// TIA Portal project "GateTest" (V17)

(* hardware
DEVICE "HMI_1"  KTP400 Comfort
   slot 0: "HMI_1"  KTP400 Comfort  6AV2 124-2DC01-0AX0  17.0.0.0
   slot 1: "HMI_RT_1"  KTP400 Comfort  6AV2 124-2DC01-0AX0  17.0.0.0
   slot 5: "HMI_1.IE_CP_1"  PROFINET Interface  17.0.0.0
      slot 1: "PROFINET Interface_1"  PROFINET Interface
         slot 1: "Port_1"  Port
   slot 7: "HMI_1.MPI/DP_CP_1"  MPI/DP Interface  17.0.0.0
DEVICE "S7-1200 station_1"  S7-1200 Station
   slot 0: "Rack_0"  S7-1200 Rack  Rack  V1.0
   slot 1: "PLC_1"  CPU 1211C DC/DC/Rly  6ES7 211-1HE40-0XB0  V4.5
   slot 101: "CM 1241 (RS422/485)_1"  6ES7 241-1CH32-0XB0  V2.2
*)

// ===== PLC "PLC_1"  CPU 1211C DC/DC/Rly =====

VAR_GLOBAL   // PLC tag table "Default tag table"
   "System_Byte" AT %MB1 : Byte;
   "FirstScan" AT %M1.0 : Bool;
   "DiagStatusUpdate" AT %M1.1 : Bool;
   "AlwaysTRUE" AT %M1.2 : Bool;
   "AlwaysFALSE" AT %M1.3 : Bool;
   "Clock_Byte" AT %MB0 : Byte;
   "Clock_10Hz" AT %M0.0 : Bool;
   "Clock_5Hz" AT %M0.1 : Bool;
   "Clock_2.5Hz" AT %M0.2 : Bool;
   "Clock_2Hz" AT %M0.3 : Bool;
   "Clock_1.25Hz" AT %M0.4 : Bool;
   "Clock_1Hz" AT %M0.5 : Bool;
   "Clock_0.625Hz" AT %M0.6 : Bool;
   "Clock_0.5Hz" AT %M0.7 : Bool;
   "IHM_Sens_Droite" AT %M2.0 : Bool;
   "IHM_Sens_Gauche" AT %M2.1 : Bool;
   "SensDroite" AT %Q0.0 : Bool;
   "SensGauche" AT %Q0.1 : Bool;
   "Busy" AT %M10.0 : Bool;
   "IHM_REQ" AT %M2.2 : Bool;
   "NB_ENTREE" AT %MW30 : Int;
   "NB_SORTIE" AT %MW32 : Int;
   "NB_INTERIEUR" AT %MW34 : Int;
   "Registre" AT %MW36 : UInt;
END_VAR

DATA_BLOCK "Data_block_1"   // DB3
{ S7_Optimized_Access := 'FALSE' }
VERSION : 0.1
   VAR
      ResultREQ : Array[0..4] of UInt;
      Registre : UInt := 40001;
      Mode : Int := 0;
   END_VAR
BEGIN
END_DATA_BLOCK

FUNCTION "CommandeMoteur" : Void   // FC1, LAD
{ S7_Optimized_Access := 'TRUE' }
VERSION : 0.1
BEGIN

REGION Network 1
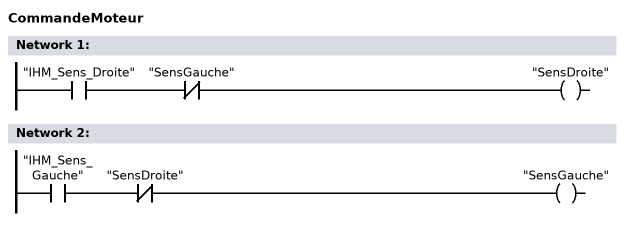
   RUNG wire#powerrail
      Contact( "IHM_Sens_Droite" )
      I_Contact( "SensGauche" )
      Coil( "SensDroite" )
   END_RUNG
   // the same network as SCL:
   "SensDroite" := "IHM_Sens_Droite" AND NOT "SensGauche";
END_REGION

REGION Network 2
   RUNG wire#powerrail
      Contact( "IHM_Sens_Gauche" )
      I_Contact( "SensDroite" )
      Coil( "SensGauche" )
   END_RUNG
   // the same network as SCL:
   "SensGauche" := "IHM_Sens_Gauche" AND NOT "SensDroite";
END_REGION
END_FUNCTION

FUNCTION "CommRS485" : Void   // FC2, LAD
{ S7_Optimized_Access := 'TRUE' }
VERSION : 0.1
BEGIN

REGION Network 1
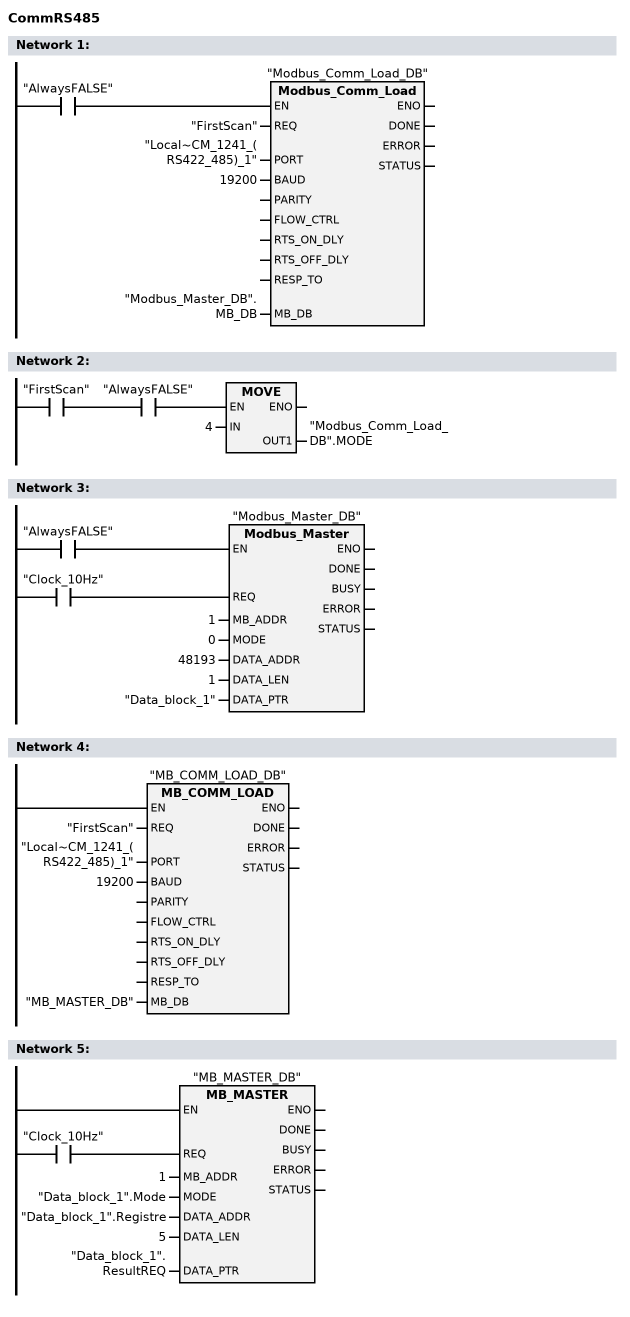
   IF "AlwaysFALSE" THEN
       "Modbus_Comm_Load_DB"(REQ := "FirstScan",   // Modbus_Comm_Load
                             PORT := "Local~CM_1241_(RS422_485)_1",
                             BAUD := 19200,
                             MB_DB := "Modbus_Master_DB".MB_DB);
   END_IF;
END_REGION

REGION Network 2
   RUNG wire#powerrail
      Contact( "FirstScan" )
      Contact( "AlwaysFALSE" )
      Move(in := 4, out1 => "Modbus_Comm_Load_DB".MODE)
   END_RUNG
   // the same network as SCL:
   IF "FirstScan" AND "AlwaysFALSE" THEN "Modbus_Comm_Load_DB".MODE := 4; END_IF;
END_REGION

REGION Network 3
   IF "AlwaysFALSE" THEN
       "Modbus_Master_DB"(REQ := "Clock_10Hz",   // Modbus_Master
                          MB_ADDR := 1,
                          MODE := 0,
                          DATA_ADDR := 48193,
                          DATA_LEN := 1,
                          DATA_PTR := "Data_block_1");
   END_IF;
END_REGION

REGION Network 4
   "MB_COMM_LOAD_DB"(REQ := "FirstScan",   // MB_COMM_LOAD
                     PORT := "Local~CM_1241_(RS422_485)_1",
                     BAUD := 19200,
                     MB_DB := "MB_MASTER_DB");
END_REGION

REGION Network 5
   "MB_MASTER_DB"(REQ := "Clock_10Hz",   // MB_MASTER
                  MB_ADDR := 1,
                  MODE := "Data_block_1".Mode,
                  DATA_ADDR := "Data_block_1".Registre,
                  DATA_LEN := 5,
                  DATA_PTR := "Data_block_1".ResultREQ);
END_REGION
END_FUNCTION

ORGANIZATION_BLOCK "Main"   // OB1, LAD, ProgramCycle
TITLE = "Main Program Sweep (Cycle)"
{ S7_Optimized_Access := 'TRUE' }
VERSION : 0.1
   VAR_INPUT
      Initial_Call : Bool;   // Initial call of this OB
      Remanence : Bool;   // =True, if remanent data are available
   END_VAR
BEGIN

REGION Network 1: Commande du moteur
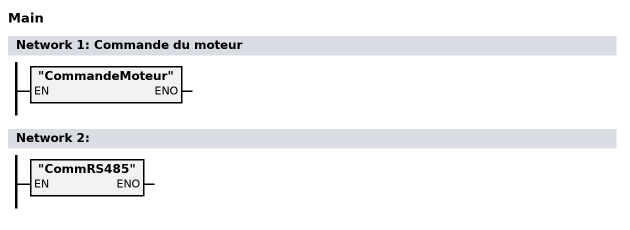
   RUNG wire#powerrail
      "CommandeMoteur"()
   END_RUNG
   // the same network as SCL:
   "CommandeMoteur"();
END_REGION

REGION Network 2
   RUNG wire#powerrail
      "CommRS485"()
   END_RUNG
   // the same network as SCL:
   "CommRS485"();
END_REGION
END_ORGANIZATION_BLOCK

(* ===== HMI "HMI_RT_1" =====
system functions are stored by id; their names below are inferred from use
connection "HMI_Connection_1": ETHERNET, S7_1200_OMS

HMI tags "Default tag table"
   "IHM_Sens_Droite" : Bool = PLC IHM_Sens_Droite AT %M2.0, 1 s
   "IHM_Sens_Gauche" : Bool = PLC IHM_Sens_Gauche AT %M2.1, 1 s
   "IHM_REQ" : Bool = PLC IHM_REQ AT %M2.2, 1 s

Template "Template_1" 480x272
   Button "Template_Button" at 415,1 size 63x63; TextOff 'Text'
   Button "Template_Button_1" at 415,70 size 63x63; TextOff 'Text'
   Button "Template_Button_2" at 415,138 size 63x63; TextOff 'Text'
   Button "Template_Button_3" at 415,207 size 63x63; TextOff 'Text'

screen "Root screen" 480x272, template "Template_1"
   TextField "HmiScreenItemData" at 42,122 size 332x22; Text 'Text'
   Button "Button_1" at 23,21 size 96x32; TextOff 'Droite'
      on Press: function_b14e0dd5("IHM_Sens_Droite", 0)
   Button "Button_2" at 278,21 size 96x32; TextOff 'Gauche'
      on Press: function_b14e0dd5("IHM_Sens_Gauche", 0)
   Button "Button_3" at 152,185 size 96x32; TextOff 'REQ'
      on Press: function_b14e0dd5("IHM_REQ", 0)
*)